TYPE ST_AssertResult :
STRUCT
    Expected          : U_ExpectedOrActual;
    ExpectedTypeClass : IBaseLibrary.TypeClass;
    Actual            : U_ExpectedOrActual;
    ActualTypeClass   : IBaseLibrary.TypeClass;
    Message           : T_MaxString;
    TestInstancePath  : T_MaxString;
END_STRUCT
END_TYPE

(* stored: Version 1.1.0.1
   DUT ST_AssertResult: Id {63e20a3e-c451-4aff-a3c2-cc9b3a584290} *)
